FUNCTION_BLOCK Conveyor_Photoeyes_Model (* Basic Function Block Type *)
  (* Standard: 61499-2 *)
  (* Version 0.0, 2010-11-05, Gareth, nxtControl GmbH, Template *)
  (* Compiler header: package fb.rt.cs725; import java.lang.Math; *)
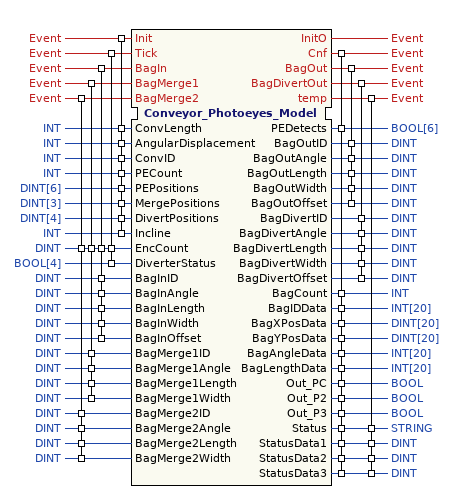
  EVENT_INPUT
    Init WITH ConvLength, AngularDisplacement, ConvID, PECount, PEPositions, MergePositions, DivertPositions, Incline; (* Initialization Request *)
    Tick WITH EncCount, DiverterStatus; (* Normal Execution Request *)
    BagIn WITH EncCount, BagInID, BagInAngle, BagInLength, BagInWidth, BagInOffset;
    BagMerge1 WITH EncCount, BagMerge1ID, BagMerge1Angle, BagMerge1Length, BagMerge1Width;
    BagMerge2 WITH EncCount, BagMerge2ID, BagMerge2Angle, BagMerge2Length, BagMerge2Width;
  END_EVENT
  EVENT_OUTPUT
    InitO; (* Initialization Confirm *)
    Cnf WITH PEDetects, BagCount, BagIDData, BagXPosData, BagYPosData, BagAngleData, BagLengthData, Out_PC, Out_P2, Out_P3, Status, StatusData1, StatusData2, StatusData3; (* Execution Confirmation *)
    BagOut WITH BagOutID, BagOutAngle, BagOutLength, BagOutWidth, BagOutOffset;
    BagDivertOut WITH BagDivertID, BagDivertAngle, BagDivertLength, BagDivertWidth, BagDivertOffset;
    temp WITH Status, StatusData1, StatusData2, StatusData3;
  END_EVENT
  VAR_INPUT
    ConvLength : INT; (* Currently in px, later in mm *)
    AngularDisplacement : INT;
    ConvID : INT;
    PECount : INT;
    PEPositions : ARRAY [0..5] OF DINT;
    MergePositions : ARRAY [0..2] OF DINT;
    DivertPositions : ARRAY [0..3] OF DINT;
    Incline : INT;
    EncCount : DINT;
    DiverterStatus : ARRAY [0..3] OF BOOL;
    BagInID : DINT;
    BagInAngle : DINT;
    BagInLength : DINT;
    BagInWidth : DINT;
    BagInOffset : DINT; (* Needed when diverting in *)
    BagMerge1ID : DINT;
    BagMerge1Angle : DINT;
    BagMerge1Length : DINT;
    BagMerge1Width : DINT;
    BagMerge2ID : DINT;
    BagMerge2Angle : DINT;
    BagMerge2Length : DINT;
    BagMerge2Width : DINT;
  END_VAR
  VAR_OUTPUT
    PEDetects : ARRAY [0..5] OF BOOL; (* Output event qualifier *)
    BagOutID : DINT;
    BagOutAngle : DINT;
    BagOutLength : DINT;
    BagOutWidth : DINT;
    BagOutOffset : DINT;
    BagDivertID : DINT;
    BagDivertAngle : DINT;
    BagDivertLength : DINT;
    BagDivertWidth : DINT;
    BagDivertOffset : DINT;
    BagCount : INT;
    BagIDData : ARRAY [0..19] OF INT;
    BagXPosData : ARRAY [0..19] OF DINT;
    BagYPosData : ARRAY [0..19] OF DINT;
    BagAngleData : ARRAY [0..19] OF INT;
    BagLengthData : ARRAY [0..19] OF INT;
    Out_PC : BOOL;
    Out_P2 : BOOL;
    Out_P3 : BOOL;
    Status : STRING;
    StatusData1 : DINT;
    StatusData2 : DINT;
    StatusData3 : DINT;
  END_VAR
  VAR
    ModelHeadPtr : INT;
    ModelTailPtr : INT;
    looper : INT;
    ModelDSPtr : INT;
    BagExited : BOOL;
    BagDiverted : BOOL;
    BagModelLLCID : ARRAY [0..19] OF DINT;
    BagModelPLCTrackStatus : ARRAY [0..19] OF INT;
    BagModelBagLength : ARRAY [0..19] OF DINT;
    BagRemoveModelPtr : INT; (* Which index to remove *)
    ConvRadius : REAL;
    currentBagAngle : ARRAY [0..19] OF REAL; (* Angle that the tangent of the curve makes with the positve x-axis *)
    BagModelBagAngle : ARRAY [0..19] OF DINT; (* Angular displacement of the bag around its center relative to the tangent to the curve *)
    BagModelBagCenterX : ARRAY [0..19] OF DINT; (* x-position of bag center *)
    BagModelBagCenterY : ARRAY [0..19] OF DINT; (* y-position of bag center *)
    BagModelBagWidth : ARRAY [0..19] OF DINT; (* width of bag *)
    BagModelBagScalarProj : ARRAY [0..19] OF DINT; (* Scalar projection magintude of the point bagCenter to the most DS point of the bag onto the x-axis *)
    BagModelBagCenterXT : ARRAY [0..19] OF DINT; (* Transformed x-position of the bag *)
    BagModelBagCenterYT : ARRAY [0..19] OF DINT; (* Transformed y-position of the bag *)
  END_VAR
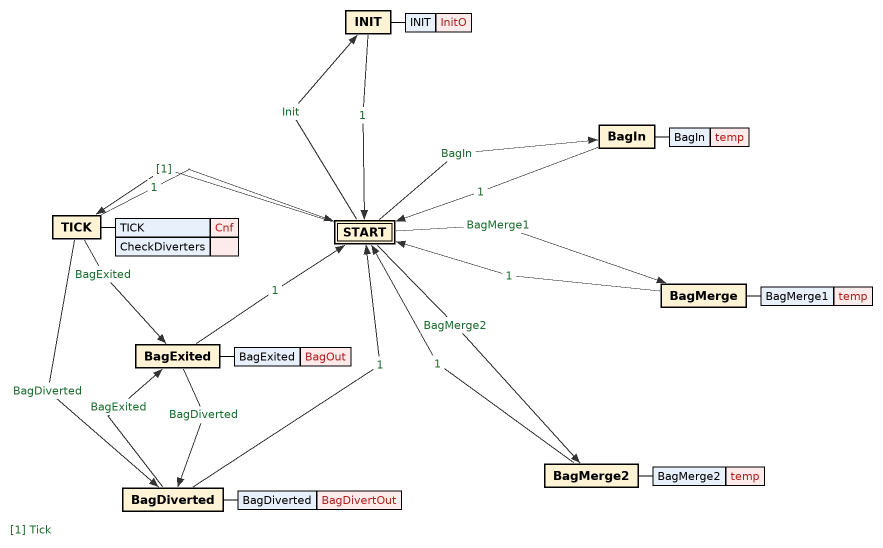
  EC_STATES
    START; (* Initial State *)
    INIT : INIT -> InitO; (* Initialization *)
    TICK : TICK -> Cnf, CheckDiverters; (* Normal execution *)
    BagIn : BagIn -> temp;
    BagMerge : BagMerge1 -> temp;
    BagExited : BagExited -> BagOut;
    BagDiverted : BagDiverted -> BagDivertOut;
    BagMerge2 : BagMerge2 -> temp;
  END_STATES
  EC_TRANSITIONS
    START TO INIT := Init;
    INIT TO START := 1;
    START TO TICK := Tick;
    BagIn TO START := 1;
    BagMerge TO START := 1;
    BagExited TO BagDiverted := BagDiverted;
    BagDiverted TO BagExited := BagExited;
    BagExited TO START := 1;
    BagDiverted TO START := 1;
    TICK TO BagExited := BagExited;
    TICK TO BagDiverted := BagDiverted;
    START TO BagIn := BagIn;
    START TO BagMerge := BagMerge1;
    TICK TO START := 1;
    START TO BagMerge2 := BagMerge2;
    BagMerge2 TO START := 1;
  END_TRANSITIONS
  ALGORITHM INIT IN Java: (* Initialization algorithm *)
ModelHeadPtr.value=(short)(0);
ModelTailPtr.value=(short)(0);
ModelDSPtr.value=(short)(-1);

for(looper.value=(short)(0); looper.value<=19; looper.value++){
((INT)BagModelPLCTrackStatus.value[looper.value]).value=(short)(0);
};


//TempPEPositions[0]).value=(short)(4500);
//TempPEPositions[1]).value=(short)(2500);
//TempPEPositions[2]).value=(short)(1500);

if((AngularDisplacement.value!=0)){
ConvRadius.value=(((ConvLength.value)*360)/(float)(2*3.14*(Math.abs((int)AngularDisplacement.value))));
};

System.out.println("Conveyor Photoeyes Initialised");
  END_ALGORITHM
  ALGORITHM TICK IN Java: (* Normally executed algorithm *)
//System.out.println("In Tick");
INT index = new INT();
INT bagPtr =  new INT();
INT upperLimit = new INT();
INT pePtr = new INT();
DINT tempOrd = new DINT();//ULINTtempOrdinateof'current'PE|diverter(EncCount.value-Position)(seeCheckDivertfor(explination)
INT CopySourcePtr = new INT();
INT CopyDestPtr = new INT();

DINT tempMostDS = new DINT();
DINT tempMostUS = new DINT();
DINT tempCount = new DINT();


bagPtr.value=ModelTailPtr.value;
upperLimit.value=ModelHeadPtr.value;

pePtr.value=0; // Pointerin((DINT)PEPositions.valueARRAY
tempOrd.value=0;

//CLEAROUTPUTS
BagExited.value=false;
BagDiverted.value=false;
BagOutID.value=(int)(0);
BagOutLength.value=(int)(0);
BagDivertID.value=(int)(0);
BagDivertLength.value=(int)(0);
//ClearDetects!!!!!!!
((BOOL)PEDetects.value[0]).value=true;
((BOOL)PEDetects.value[1]).value=true;
((BOOL)PEDetects.value[2]).value=true;
((BOOL)PEDetects.value[3]).value=true;
((BOOL)PEDetects.value[4]).value=true;
((BOOL)PEDetects.value[5]).value=true;


//NOOOOO"Loop through all bags... increment Positions?"
//usingordinates...assumingbagsdontslipwewontneed; ModelTailPtr.value<=changetheirUS/DSOrd
if(ModelTailPtr.value>ModelHeadPtr.value)
{
upperLimit.value=(short)(ModelHeadPtr.value+20); //sizeofBagARRAY
};

for(pePtr.value=0; pePtr.value<=PECount.value-1; pePtr.value++)
{
tempOrd.value=(EncCount.value-(((DINT)PEPositions.value[(int)pePtr.value]).value));
for(bagPtr.value= ModelTailPtr.value; bagPtr.value<=upperLimit.value-1; bagPtr.value++)
{
//CalculatethemostDS&USpositionofthebag
tempMostDS.value = (((DINT)(BagModelBagCenterX.value[bagPtr.value%20])).value + ((DINT)BagModelBagScalarProj.value[bagPtr.value%20]).value);
tempMostUS.value = (((DINT)BagModelBagCenterX.value[bagPtr.value %20]).value-((DINT)BagModelBagScalarProj.value[bagPtr.value%20]).value);
if((tempMostDS.value>=tempOrd.value)&(tempMostUS.value<=tempOrd.value))
{
//thisPEneeds; ModelTailPtr.value<='detect'
//((BOOL)PEDetects.value[pePtr.value]).value=true;
((BOOL)PEDetects.value[pePtr.value]).value=false;

break; //onlyonebagcanintersect...
}
}
}

/*CheckmostDSBag..if(passedConvLength....valuestartcontinueprocess
Everythingmodelledasastraightconveyor&bagstrackedusingcenterx,y+angle
TODO:if(array!EMPTY */
if((ModelDSPtr.value!=-1))
{
//Ensurethebaghas!alreadyexited
if((((INT)BagModelPLCTrackStatus.value[ModelDSPtr.value]).value==2))
{//ACTIVE
//'continue'thebagwhenthecenterofthebagreachestheendofthisconveyor
if((EncCount.value>=(((DINT)BagModelBagCenterX.value[ModelDSPtr.value]).value+ConvLength.value)))
{//>*==*soassoonascenterpointisatDS'tip',itisalsoatmostUSendofDSConv
//Status.value='Bagcenterpointexited';

//Thebaghas'exited'i.e.belongs; ModelTailPtr.value<=thenextconveyorinanobjectownershipsense
BagOutID.value=(((DINT)BagModelLLCID.value[ModelDSPtr.value]).value);
BagOutLength.value=(int)(((DINT)BagModelBagLength.value[ModelDSPtr.value]).value);
BagOutWidth.value=(int)(((DINT)BagModelBagWidth.value[ModelDSPtr.value]).value);

BagOutOffset.value=(int)(((DINT)BagModelBagCenterY.value[ModelDSPtr.value]).value);//y-axisoffset,zerofor(now
BagOutAngle.value=(int)(((DINT)BagModelBagAngle.value[ModelDSPtr.value]).value);

BagExited.value=true;
((INT)BagModelPLCTrackStatus.value[ModelDSPtr.value]).value=(short)(3);
}
}
else if((((INT)BagModelPLCTrackStatus.value[ModelDSPtr.value]).value==3))
{//COMPLETED//Centerhasexited..justwaitingonmostUSpoint
//Re-calculatethemostUSx-position
tempMostUS.value=(((DINT)BagModelBagCenterX.value[ModelDSPtr.value]).value-((DINT)BagModelBagScalarProj.value[ModelDSPtr.value]).value);
if(((EncCount.value-tempMostUS.value)>ConvLength.value))
{
//Justremovefrommodel
((INT)BagModelPLCTrackStatus.value[ModelDSPtr.value]).value=(short)(0);
/*Status.value='Bagremoved';
StatusData1.value=(int)((EncCount.value-BagModelBagUSOrd[ModelDSPtr.value]).value));*/
//ConveyorModel_CM_RemoveBag(me,((DINT)BagModelLLCID.value[ModelDSPtr.value]).value,ModelDSPtr);
CopyDestPtr.value=(short)(ModelDSPtr.value);//Overwritethisbag
while(true)
{
BagOutAngle.value++;
//IsthistheMostDSbag?
if((CopyDestPtr.value==ModelTailPtr.value))
{
//Deletethemodelentry
((DINT)BagModelLLCID.value[CopyDestPtr.value]).value=(int)(-1);
//UpdateDSpointer
ModelTailPtr.value=(short)(ModelTailPtr.value+1);
ModelTailPtr.value=(short)(ModelTailPtr.value%20);
//RE-setModelDSPtr.value
ModelDSPtr.value=(short)(-1);
//FindthemostDSbag; BagOutAngle.value<=settheModelDSPtr.value
for(bagPtr.value=(short)((ModelTailPtr.value)); bagPtr.value<=upperLimit.value-1; bagPtr.value++)
{
if((((DINT)BagModelLLCID.value[bagPtr.value]).value%20!=-1))
{
if((ModelDSPtr.value<0))
{ //thisnewbagismoreDSthanlastmostDS...shufflearray
ModelDSPtr.value=(short)(bagPtr.value%20);
}
else if(((DINT)BagModelBagCenterX.value[bagPtr.value%20]).value<((DINT)BagModelBagCenterX.value[ModelDSPtr.value]).value)
{
ModelDSPtr.value=(short)(bagPtr.value%20);
}
}
}
Status.value= (new String("TICK most DS bag")).getBytes();
break;
}
else
{
//CalculatetheCopySourcePtr
if((CopyDestPtr.value==0))
{
CopySourcePtr.value=20-1;//"Next entry is top"
}
else
{
CopySourcePtr.value=(short)((CopyDestPtr.value-1)%20);
}
//CopyModelData
((DINT)BagModelLLCID.value[CopyDestPtr.value]).value=(int)(((DINT)BagModelLLCID.value[CopySourcePtr.value]).value);
((DINT)BagModelBagLength.value[CopyDestPtr.value]).value=(int)(((DINT)BagModelBagLength.value[CopySourcePtr.value]).value);
((INT)BagModelPLCTrackStatus.value[CopyDestPtr.value]).value=(short)(((INT)BagModelPLCTrackStatus.value[CopySourcePtr.value]).value);
((DINT)BagModelBagWidth.value[CopyDestPtr.value]).value=(int)(((DINT)BagModelBagWidth.value[CopySourcePtr.value]).value);
((DINT)BagModelBagAngle.value[CopyDestPtr.value]).value=(int)(((DINT)BagModelBagAngle.value[CopySourcePtr.value]).value);
((DINT)BagModelBagCenterX.value[CopyDestPtr.value]).value=(int)(((DINT)BagModelBagCenterX.value[CopySourcePtr.value]).value);
((DINT)BagModelBagCenterY.value[CopyDestPtr.value]).value=(int)(((DINT)BagModelBagCenterY.value[CopySourcePtr.value]).value);
((DINT)BagModelBagScalarProj.value[CopyDestPtr.value]).value=(int)(((DINT)BagModelBagScalarProj.value[CopySourcePtr.value]).value);
//nextmodelentry
CopyDestPtr.value=(short)(CopySourcePtr.value);
}
}
//ENDREMOVEINLINE
upperLimit.value=(short)(ModelHeadPtr.value);//REDOupperLimit.value(mayhavechanged)
if((ModelTailPtr.value>ModelHeadPtr.value))
{
upperLimit.value=(short)(ModelHeadPtr.value+20);//sizeofBagarray
}
}
}
}
//Transformstraightconveyordisplacement; ModelTailPtr.value<=curvedconveyordisplacement
for(bagPtr.value=(short)(ModelTailPtr.value); bagPtr.value<=upperLimit.value-1; bagPtr.value++)
{
if((AngularDisplacement.value!=0))
{
((REAL)currentBagAngle.value[bagPtr.value]).value=(float)(((EncCount.value-((DINT)BagModelBagCenterX.value[bagPtr.value%20]).value)/(ConvLength.value))*(AngularDisplacement.value));
((DINT)BagModelBagCenterXT.value[bagPtr.value%20]).value=(int)((ConvRadius.value*Math.sin((((REAL)currentBagAngle.value[bagPtr.value]).value/180)*3.14)));
((DINT)BagModelBagCenterYT.value[bagPtr.value%20]).value=(int)((ConvRadius.value-ConvRadius.value*Math.cos((((REAL)currentBagAngle.value[bagPtr.value]).value/180)*3.14)));
//However,if(thebagisleavingtheconveyor,maybe){otherstuff,likegoinastraightlineafterpassingconvLength
}
else
{
/*(
else{thisisastraightline*/
((DINT)BagModelBagCenterXT.value[bagPtr.value%20]).value=(int)(EncCount.value-((DINT)BagModelBagCenterX.value[bagPtr.value%20]).value);
((DINT)BagModelBagCenterYT.value[bagPtr.value%20]).value=(int)(((DINT)BagModelBagCenterY.value[bagPtr.value%20]).value);
}
}

//SetVisData
BagCount.value=(short)(upperLimit.value-ModelTailPtr.value);
bagPtr.value=(short)(ModelTailPtr.value);
//cleararrays
for(bagPtr.value=(short)(0); bagPtr.value<=19; bagPtr.value++)
{
((INT)BagIDData.value[bagPtr.value]).value=(short)(0);
((DINT)BagXPosData.value[bagPtr.value]).value=0;
((INT)BagLengthData.value[bagPtr.value]).value=(short)(0);
}

bagPtr.value=(short)(ModelTailPtr.value);
for(index.value=(short)(0); index.value<=19; index.value++)
{
if((bagPtr.value>=upperLimit.value))
{
break;
};

((DINT)BagYPosData.value[index.value]).value=(int)(((DINT)BagModelBagCenterYT.value[bagPtr.value%20]).value);
((DINT)BagXPosData.value[index.value]).value=(int)(((DINT)BagModelBagCenterXT.value[bagPtr.value%20]).value)+1;
((INT)BagAngleData.value[index.value]).value=(short)((((REAL)currentBagAngle.value[bagPtr.value%20]).value)+(((DINT)BagModelBagAngle.value[bagPtr.value%20]).value));
((INT)BagLengthData.value[index.value]).value=(short)((((DINT)BagModelBagLength.value[bagPtr.value%20]).value));
//((INT)BagWidthData.value[index.value]).value=(short)((((DINT)BagModelBagWidth.value[bagPtr.value%20]).value));
((INT)BagIDData.value[index.value]).value=(short)((((DINT)BagModelLLCID.value[bagPtr.value%20]).value));

bagPtr.value++;
};

//Tempfixfor(non-blankingarrays
if((BagCount.value==0))
{
((DINT)BagYPosData.value[0]).value=(int)(0);
((DINT)BagXPosData.value[0]).value=0;
((INT)BagAngleData.value[0]).value=(short)(0);
((INT)BagLengthData.value[0]).value=(short)(0);
//((INT)BagWidthData.value[0]).value=(short)(0);
((INT)BagIDData.value[0]).value=(short)(0);
}

//TEMPUN-ARRAY
Out_PC.value=((BOOL)PEDetects.value[0]).value;
//System.out.println("PE SET = " + ((BOOL)PEDetects.value[0]).value + Out_PC.value);
Out_P2.value=((BOOL)PEDetects.value[1]).value;
Out_P3.value=((BOOL)PEDetects.value[2]).value;
  END_ALGORITHM
  ALGORITHM BagIn IN Java:
REAL bagRectTopRightX = new REAL();
REAL bagRectBottomRightX = new REAL();
DINT tempX = new DINT();
REAL bagRectRadius = new REAL(); //Halfthelengthofthediagonalinsidethebagrectangle
REAL bagRectInternalAngle = new REAL(); //Theanglethediagonalmakeswiththepositivex-axisofthebag

System.out.println("Bag IN!!! and ModelHeadPtr = " + ModelHeadPtr.value + " ModelDSPtr = " + ModelDSPtr.value);

if(((INT)BagModelPLCTrackStatus.value[ModelHeadPtr.value]).value==2){//ACTIVE ModelFull
return;
};

if (ModelDSPtr.value<0)
{ //thisnewbagismoreDSthanlastmostDS...
ModelDSPtr.value=(short)(ModelHeadPtr.value); //ThelocationwherethisTHINGwillbestored
}
else if ((EncCount.value-BagInOffset.value) < ((DINT)BagModelBagCenterX.value[ModelDSPtr.value]).value)
{ //thisnewbagismoreDSthanlastmostDS...
ModelDSPtr.value=(short)(ModelHeadPtr.value); //ThelocationwherethisTHINGwillbestored
}


((DINT)BagModelBagCenterX.value[ModelHeadPtr.value]).value=(int)(EncCount.value);
((DINT)BagModelBagWidth.value[ModelHeadPtr.value]).value=(int)(BagInWidth.value);
((DINT)BagModelBagCenterY.value[ModelHeadPtr.value]).value=(int)(0);
((DINT)BagModelBagAngle.value[ModelHeadPtr.value]).value=(int)(BagInAngle.value);
((DINT)BagModelLLCID.value[ModelHeadPtr.value]).value=(int)(BagInID.value);
((DINT)BagModelBagLength.value[ModelHeadPtr.value]).value=(int)(BagInLength.value);
((INT)BagModelPLCTrackStatus.value[ModelHeadPtr.value]).value=(short)(2); //ACTIVE

 //Calculatethex-distancebetweenthemostdownstreampointofthebagminusthecenterpoint
bagRectRadius.value=(float)Math.sqrt((BagInLength.value/2)*(BagInLength.value/2)+(BagInWidth.value/2)*(BagInWidth.value/2));
bagRectInternalAngle.value=(float)Math.atan(BagInWidth.value/BagInLength.value);

bagRectTopRightX.value=(bagRectRadius.value*(float)Math.cos(3.14*((((DINT)BagModelBagAngle.value[ModelHeadPtr.value]).value))/180+bagRectInternalAngle.value));
bagRectBottomRightX.value=(bagRectRadius.value*(float)Math.cos(3.14*((((DINT)BagModelBagAngle.value[ModelHeadPtr.value]).value))/180-bagRectInternalAngle.value));


if((BagInAngle.value<90)){
((DINT)BagModelBagScalarProj.value[ModelHeadPtr.value]).value=(int)(bagRectBottomRightX.value);
}
else if((BagInAngle.value<180)){
((DINT)BagModelBagScalarProj.value[ModelHeadPtr.value]).value=(int)(-1*bagRectTopRightX.value);
}
else if((BagInAngle.value<270)){
((DINT)BagModelBagScalarProj.value[ModelHeadPtr.value]).value=(int)(-1*bagRectBottomRightX.value);
}
else if((BagInAngle.value<360)){
((DINT)BagModelBagScalarProj.value[ModelHeadPtr.value]).value=(int)(bagRectTopRightX.value);
};

//Incrementthepointers
ModelHeadPtr.value=(short)(ModelHeadPtr.value+1);
ModelHeadPtr.value=(short)(ModelHeadPtr.value%20);
  END_ALGORITHM
  ALGORITHM BagMerge1 IN Java:
REAL bagRectTopRightX = new REAL();
REAL bagRectBottomRightX = new REAL();
DINT tempX = new DINT();
REAL bagRectRadius = new REAL(); //Halfthelengthofthediagonalinsidethebagrectangle
REAL bagRectInternalAngle = new REAL(); //Theanglethediagonalmakeswiththepositivex-axisofthebag

System.out.println("BagMerge1!!");

if(((INT)BagModelPLCTrackStatus.value[ModelHeadPtr.value]).value==2){ //ACTIVE ModelFull
return;
};

if(ModelDSPtr.value<0)
{
ModelDSPtr.value=(short)(ModelHeadPtr.value); //ThelocationwherethisTHINGwillbestored
Status.value= (new String("NewmostDSbag")).getBytes();;
}
else if(((EncCount.value-(((DINT)MergePositions.value[0]).value))<((DINT)BagModelBagCenterX.value[ModelDSPtr.value]).value)){ //thisnewbagismoreDSthanlastmostDS...
ModelDSPtr.value=(short)(ModelHeadPtr.value); //ThelocationwherethisTHINGwillbestored
Status.value= (new String("NewmostDSbag")).getBytes();;
};

((DINT)BagModelBagCenterX.value[ModelHeadPtr.value]).value=(int)(EncCount.value-((DINT)MergePositions.value[0]).value);
((DINT)BagModelBagWidth.value[ModelHeadPtr.value]).value=(int)(BagMerge1Width.value);
((DINT)BagModelBagCenterY.value[ModelHeadPtr.value]).value=(int)(0);
((DINT)BagModelBagAngle.value[ModelHeadPtr.value]).value=(int)(BagMerge1Angle.value);
((DINT)BagModelLLCID.value[ModelHeadPtr.value]).value=(int)(BagMerge1ID.value);
((DINT)BagModelBagLength.value[ModelHeadPtr.value]).value=(int)(BagMerge1Length.value);
((INT)BagModelPLCTrackStatus.value[ModelHeadPtr.value]).value=(short)(2); //ACTIVE

//Calculatethex-distancebetweenthemostdownstreampointofthebagminusthecenterpoint
bagRectRadius.value= (float)Math.sqrt(((BagMerge1Length.value/2)*(BagMerge1Length.value/2))+((BagMerge1Width.value/2)*(BagMerge1Width.value/2)));
bagRectInternalAngle.value=(float)Math.atan(BagMerge1Width.value/BagMerge1Length.value);

bagRectTopRightX.value=(bagRectRadius.value*(float)Math.cos(3.14*((((DINT)BagModelBagAngle.value[ModelHeadPtr.value]).value))/180+bagRectInternalAngle.value));
bagRectBottomRightX.value=(bagRectRadius.value*(float)Math.cos(3.14*((((DINT)BagModelBagAngle.value[ModelHeadPtr.value]).value))/180-bagRectInternalAngle.value));

if((BagInAngle.value<90)){
((DINT)BagModelBagScalarProj.value[ModelHeadPtr.value]).value=(int)(bagRectBottomRightX.value);
}
else if((BagInAngle.value<180)){
((DINT)BagModelBagScalarProj.value[ModelHeadPtr.value]).value=(int)(-1*bagRectTopRightX.value);
}
else if((BagInAngle.value<270)){
((DINT)BagModelBagScalarProj.value[ModelHeadPtr.value]).value=(int)(-1*bagRectBottomRightX.value);
}
else if((BagInAngle.value<360)){
((DINT)BagModelBagScalarProj.value[ModelHeadPtr.value]).value=(int)(bagRectTopRightX.value);
};

//Increment
ModelHeadPtr.value=(short)(ModelHeadPtr.value+1);
ModelHeadPtr.value=(short)(ModelHeadPtr.value%20);
  END_ALGORITHM
  ALGORITHM CheckDiverters IN Java:
INT upperLimit = new INT();
INT bagPtr = new INT();
INT DivID = new INT();
DINT tempOrd = new DINT(); //ULINT
INT CopySourcePtr = new INT();
INT CopyDestPtr = new INT();

//System.out.println("In CheckDiverters");

DINT tempMostDS = new DINT();
DINT tempMostUS = new DINT();


upperLimit.value=ModelHeadPtr.value;
DivID.value=0;
/*
EncCount.value-BagOrd=(int)(Position
|
EncCount.value-Position=(int)(BagOrd
(sowegetEncCount.value-PosONCE..&comparewithbagords)
*/
tempOrd.value=0;// Special*ORDINATEofdiverter(EncCount.value-Position)
/*//if(thediverterisactive
checkupperLimit*/
if(((ModelHeadPtr.value)<(ModelTailPtr.value)))
{
upperLimit.value=(short)(upperLimit.value+20);//Lengthofbagarray
}

while(DivID.value<4)
{
if((((DINT)DivertPositions.value[DivID.value]).value>0&((BOOL)DiverterStatus.value[DivID.value]).value))
{//configured&'active'//Statuses+1becauseitalsocontainsExitDev0whichisrunout
tempOrd.value=EncCount.value-((DINT)DivertPositions.value[DivID.value]).value;
//Anybagsthatintersect/cross'DiverterPosition'isdiverted(assumeonlyonebagperanyONEtick)
for(bagPtr.value=(short)((ModelTailPtr.value)); bagPtr.value<=upperLimit.value-1; bagPtr.value++)
{
//CalculatethemostDS&USpositionofthebag
tempMostDS.value=(((DINT)BagModelBagCenterX.value[bagPtr.value%20]).value+((DINT)BagModelBagScalarProj.value[bagPtr.value%20]).value);
tempMostUS.value=(((DINT)BagModelBagCenterX.value[bagPtr.value%20]).value-((DINT)BagModelBagScalarProj.value[bagPtr.value%20]).value);

if(((tempMostUS.value>=tempOrd.value)&(tempMostDS.value<=tempOrd.value)))
{
/*thisBagINTERSECTS!!!
setaflag*///
BagDiverted.value=true;
BagDivertID.value=(int)(((DINT)BagModelLLCID.value[bagPtr.value%20]).value);
BagDivertLength.value=(int)(((DINT)BagModelBagLength.value[bagPtr.value%20]).value);
//2010-07-05:HandoverOffset(howfarINFRONTofDiverterthebagis)
BagDivertOffset.value=(int)(tempOrd.value-((DINT)BagModelBagCenterX.value[bagPtr.value%20]).value);
//Unlikenormalexit...weIMEDIATELYremovethebagfromourmodel(itwill!passanymorePEs)
//ConveyorModel_CM_RemoveBag(me,BagDivertID,bagPtr.value%20);
CopyDestPtr.value=(short)(bagPtr.value%20);//Overwritethisbag
while(true)
{
//IsthistheMostDSbag?
if((CopyDestPtr.value==ModelTailPtr.value))
{
//Deletethemodelentry
((DINT)BagModelLLCID.value[CopyDestPtr.value]).value=(int)(-1);
//UpdateDSpointer
ModelTailPtr.value=(short)(ModelTailPtr.value+1);
ModelTailPtr.value=(short)(ModelTailPtr.value%20);
//RE-setModelDSPtr.value
ModelDSPtr.value=(short)(-1);
for(bagPtr.value=(short)((ModelTailPtr.value)); bagPtr.value<=upperLimit.value-1; bagPtr.value++)
{
if((((DINT)BagModelLLCID.value[bagPtr.value]).value%20!=-1))
{
if((ModelDSPtr.value<0))
{//thisnewbagismoreDSthanlastmostDS...shufflearray
ModelDSPtr.value=(short)(bagPtr.value%20);
}
else if(((DINT)BagModelBagCenterX.value[bagPtr.value%20]).value<((DINT)BagModelBagCenterX.value[ModelDSPtr.value]).value)
{
ModelDSPtr.value=(short)(bagPtr.value%20);
}
}
}
break;
}
else
{
//CalculatetheCopySourcePtr
if((CopyDestPtr.value==0))
{
CopySourcePtr.value=20-1;//"Next entry is top"
}
else
{
CopySourcePtr.value=(short)((CopyDestPtr.value-1)%20);
}

//CopyModelData
((DINT)BagModelLLCID.value[CopyDestPtr.value]).value=(int)(((DINT)BagModelLLCID.value[CopySourcePtr.value]).value);
((DINT)BagModelBagLength.value[CopyDestPtr.value]).value=(int)(((DINT)BagModelBagLength.value[CopySourcePtr.value]).value);
((INT)BagModelPLCTrackStatus.value[CopyDestPtr.value]).value=(short)(((INT)BagModelPLCTrackStatus.value[CopySourcePtr.value]).value);
((DINT)BagModelBagWidth.value[CopyDestPtr.value]).value=(int)(((DINT)BagModelBagWidth.value[CopySourcePtr.value]).value);
((DINT)BagModelBagAngle.value[CopyDestPtr.value]).value=(int)(((DINT)BagModelBagAngle.value[CopySourcePtr.value]).value);
((DINT)BagModelBagCenterX.value[CopyDestPtr.value]).value=(int)(((DINT)BagModelBagCenterX.value[CopySourcePtr.value]).value);
((DINT)BagModelBagCenterY.value[CopyDestPtr.value]).value=(int)(((DINT)BagModelBagCenterY.value[CopySourcePtr.value]).value);
((DINT)BagModelBagScalarProj.value[CopyDestPtr.value]).value=(int)(((DINT)BagModelBagScalarProj.value[CopySourcePtr.value]).value);
//nextmodelentry
CopyDestPtr.value=CopySourcePtr.value;
}
}
break;
}
}
}
DivID.value++;
}
  END_ALGORITHM
  ALGORITHM RemoveBag IN Java:
INT CopySourcePtr = new INT();
INT CopyDestPtr = new INT();
INT bagPtr = new INT();
DINT upperBound = new DINT();//ULINT

CopySourcePtr.value=-1;
CopyDestPtr.value=-1;
upperBound.value=ModelHeadPtr.value;

if((ModelHeadPtr.value<ModelTailPtr.value))
{
upperBound.value=(short)(upperBound.value+20);
}

CopyDestPtr.value=(short)(BagRemoveModelPtr.value);//Overwritethisbag
if((CopyDestPtr.value==-1))
{
return;
}


while(true)
{
//IsthistheMostDSbag?
if((CopyDestPtr.value==ModelTailPtr.value))
{
//Deletethemodelentry
((DINT)BagModelLLCID.value[CopyDestPtr.value]).value=(int)(-1);
//UpdateDSpointer
ModelTailPtr.value=(short)(ModelTailPtr.value+1);
ModelTailPtr.value=(short)(ModelTailPtr.value%20);
//RE-setModelDSPtr.value
ModelDSPtr.value=(short)(-1);
for(bagPtr.value=(short)((ModelTailPtr.value)); bagPtr.value<=upperBound.value; bagPtr.value++)
{
if((((DINT)BagModelLLCID.value[bagPtr.value]).value%20!=-1))
{
if((ModelDSPtr.value<0))
{//thisnewbagismoreDSthanlastmostDS...shufflearray
ModelDSPtr.value=(short)(bagPtr.value%20);
}
else if(((DINT)BagModelBagCenterX.value[bagPtr.value%20]).value<((DINT)BagModelBagCenterX.value[ModelDSPtr.value]).value)
{
ModelDSPtr.value=(short)(bagPtr.value%20);
}
}
}
break;
}
else
{
//CalculatetheCopySourcePtr
if((CopyDestPtr.value==0))
{
CopySourcePtr.value=(short)(20-1);//"Next entry is top"
}
else
{
CopySourcePtr.value=(short)((CopyDestPtr.value-1)%20);
}
//CopyModelData
((DINT)BagModelLLCID.value[CopyDestPtr.value]).value=(int)(((DINT)BagModelLLCID.value[CopySourcePtr.value]).value);
((DINT)BagModelBagLength.value[CopyDestPtr.value]).value=(int)(((DINT)BagModelBagLength.value[CopySourcePtr.value]).value);
((INT)BagModelPLCTrackStatus.value[CopyDestPtr.value]).value=(short)(((INT)BagModelPLCTrackStatus.value[CopySourcePtr.value]).value);
((DINT)BagModelBagWidth.value[CopyDestPtr.value]).value=(int)(((DINT)BagModelBagWidth.value[CopySourcePtr.value]).value);
((DINT)BagModelBagAngle.value[CopyDestPtr.value]).value=(int)(((DINT)BagModelBagAngle.value[CopySourcePtr.value]).value);
((DINT)BagModelBagCenterX.value[CopyDestPtr.value]).value=(int)(((DINT)BagModelBagCenterX.value[CopySourcePtr.value]).value);
((DINT)BagModelBagCenterY.value[CopyDestPtr.value]).value=(int)(((DINT)BagModelBagCenterY.value[CopySourcePtr.value]).value);
((DINT)BagModelBagScalarProj.value[CopyDestPtr.value]).value=(int)(((DINT)BagModelBagScalarProj.value[CopySourcePtr.value]).value);

//nextmodelentry
CopyDestPtr.value=(short)(CopySourcePtr.value);
}
}
  END_ALGORITHM
  ALGORITHM BagExited IN Java:
BagExited.value=false;//DONE
System.out.println("BagOut!!");
  END_ALGORITHM
  ALGORITHM BagDiverted IN Java:
BagDiverted.value=false; //DONE
  END_ALGORITHM
  ALGORITHM BagMerge2 IN Java:
REAL bagRectTopRightX = new REAL();
REAL bagRectBottomRightX = new REAL();
DINT tempX = new DINT();;
REAL bagRectRadius = new REAL();;//Halfthelengthofthediagonalinsidethebagrectangle
REAL bagRectInternalAngle = new REAL();;//Theanglethediagonalmakeswiththepositivex-axisofthebag

System.out.println("BagMerge2!!");
if(((INT)BagModelPLCTrackStatus.value[ModelHeadPtr.value]).value==2){//ACTIVE ModelFull
return;
};

if(ModelDSPtr.value<0)
{
ModelDSPtr.value=(short)(ModelHeadPtr.value);//ThelocationwherethisTHINGwillbestored
Status.value=(new String("NewmostDSbag")).getBytes();
}
else if (((EncCount.value-((DINT)MergePositions.value[1]).value)<((DINT)BagModelBagCenterX.value[ModelDSPtr.value]).value)){//thisnewbagismoreDSthanlastmostDS...
ModelDSPtr.value=(short)(ModelHeadPtr.value);//ThelocationwherethisTHINGwillbestored
Status.value=(new String("NewmostDSbag")).getBytes();
};

((DINT)BagModelBagCenterX.value[ModelHeadPtr.value]).value=(int)(EncCount.value-((DINT)MergePositions.value[1]).value);
((DINT)BagModelBagWidth.value[ModelHeadPtr.value]).value=(int)(BagMerge2Width.value);
((DINT)BagModelBagCenterY.value[ModelHeadPtr.value]).value=(int)(0);
((DINT)BagModelBagAngle.value[ModelHeadPtr.value]).value=(int)(BagMerge2Angle.value);
((DINT)BagModelLLCID.value[ModelHeadPtr.value]).value=(int)(BagMerge2ID.value);
((DINT)BagModelBagLength.value[ModelHeadPtr.value]).value=(int)(BagMerge2Length.value);
((INT)BagModelPLCTrackStatus.value[ModelHeadPtr.value]).value=(short)(2);//ACTIVE

//Calculatethex-distancebetweenthemostdownstreampointofthebagminusthecenterpoint
bagRectRadius.value= (float)Math.sqrt(((BagMerge2Length.value/2)*(BagMerge2Length.value/2))+((BagMerge2Width.value/2)*(BagMerge2Width.value/2)));
bagRectInternalAngle.value=(float)Math.atan(BagMerge2Width.value/BagMerge2Length.value);

bagRectTopRightX.value=(bagRectRadius.value*(float)Math.cos(3.14*((((DINT)BagModelBagAngle.value[ModelHeadPtr.value]).value))/180+bagRectInternalAngle.value));
bagRectBottomRightX.value=(bagRectRadius.value*(float)Math.cos(3.14*((((DINT)BagModelBagAngle.value[ModelHeadPtr.value]).value))/180-bagRectInternalAngle.value));

if((BagInAngle.value<90)){
((DINT)BagModelBagScalarProj.value[ModelHeadPtr.value]).value=(int)((bagRectBottomRightX.value));
}
else if((BagInAngle.value<180)){
((DINT)BagModelBagScalarProj.value[ModelHeadPtr.value]).value=(int)((-1*bagRectTopRightX.value));
}
else if((BagInAngle.value<270)){
((DINT)BagModelBagScalarProj.value[ModelHeadPtr.value]).value=(int)((-1*bagRectBottomRightX.value));
}
else if((BagInAngle.value<360)){
((DINT)BagModelBagScalarProj.value[ModelHeadPtr.value]).value=(int)((bagRectTopRightX.value));
};

//Increment
ModelHeadPtr.value=(short)(ModelHeadPtr.value+1);
ModelHeadPtr.value=(short)(ModelHeadPtr.value%20);
  END_ALGORITHM
END_FUNCTION_BLOCK
